Fanuc KAREL source: SAVE_DRAM.kl

PROGRAM T
%NOLOCKGROUP
VAR
 v0 : STRING[40]
 v1 : INTEGER
BEGIN
 SAVE_DRAM(v0, v1)
END T
